FUNCTION_BLOCK FB_ConveyorPeerSequence IMPLEMENTS I_ConveyorSequence
VAR_INPUT

END_VAR
VAR_OUTPUT
END_VAR
VAR
	nStep : E_ConveyorPeerSequence;
END_VAR

METHOD M_ConveyorAction : BOOL
VAR_INPUT
	in_stFirstMessage : ST_Message;
	in_stMessageToCheckFor : ST_Message;
	in_stSecondMessage : ST_Message;
	in_rConveyor : REFERENCE TO FB_Conveyor;
END_VAR
VAR_INST
	nConveyorActionStep : UINT;
END_VAR
CASE nConveyorActionStep OF
	
	0:
		IF 	in_rConveyor.M_SendMessage
			(	
				in_stFirstMessage
			) 
			= E_PeerReturnCode.eMESSAGE_IN_OUTBOX 
			THEN
			
			nConveyorActionStep := 10;
			
		END_IF
		
	10:
		
	
		IF 	in_rConveyor.M_CompareMessageAndEmptyMailbox
			(	
				in_stMessageToCheckFor
			) 
			= E_PeerReturnCode.eMATCH_FOUND 
			THEN
			
			nConveyorActionStep := 20;
			
		END_IF

	20:
		
		IF 	in_rConveyor.M_SendMessage
			(	
				in_stSecondMessage
			) 
			= E_PeerReturnCode.eMESSAGE_IN_OUTBOX 
			THEN
			
			nConveyorActionStep := 0;
			M_ConveyorAction := TRUE;
			
		END_IF
		
END_CASE
END_METHOD


METHOD M_ConveyorSequence : BOOL
VAR_INPUT
	in_rConveyor : REFERENCE TO FB_Conveyor;
END_VAR
CASE nStep OF
	
	E_ConveyorPeerSequence.eSTOP:
	
		nStep := E_ConveyorPeerSequence.eSTART;
		
	E_ConveyorPeerSequence.eSTART:
		
		in_rConveyor.M_StartConveyor();
		nStep := E_ConveyorPeerSequence.eSTOP_AT_SIGNAL;

	E_ConveyorPeerSequence.eSTOP_AT_SIGNAL:
	
		IF in_rConveyor.out_fbSensorStop.GetSignal THEN
			in_rConveyor.M_StopConveyor();
			nStep := E_ConveyorPeerSequence.eWAIT_FOR_ACK;
		END_IF
	
	E_ConveyorPeerSequence.eWAIT_FOR_ACK:
		
		IF M_SubjectiveAction(in_rConveyor) THEN
			nStep := E_ConveyorPeerSequence.eRESUME_OPERATION;
		END_IF
	
	E_ConveyorPeerSequence.eRESUME_OPERATION:
		
		in_rConveyor.M_StartConveyor();
		IF in_rConveyor.out_fbSensorMaterialDispatch.GetSignal THEN
			in_rConveyor.M_StopConveyor();
			nStep := E_ConveyorPeerSequence.eEND_SEQUENCE;
		END_IF
	
	E_ConveyorPeerSequence.eEND_SEQUENCE:
		;
		
END_CASE
END_METHOD

METHOD M_Sequence : BOOL
VAR_INPUT
END_VAR
END_METHOD

METHOD M_SubjectiveAction : BOOL
VAR_INPUT
	in_rConveyor : REFERENCE TO FB_Conveyor;
END_VAR
CASE in_rConveyor.M_GetPeerId() OF

	E_PeersList.ePEER_CONVEYOR_1:
		
		IF 	M_ConveyorAction
			(
				Message(eCONVEYOR_1_AT_TRANSFER_POINT,ePEER_CONVEYOR_2),
				Message(eCONVEYOR_4_AT_TRANSFER_POINT,ePEER_CONVEYOR_4),
 				Message(eCONVEYOR_1_RESUMING_OPERATION,ePEER_CONVEYOR_2),
				in_rConveyor
			) 
			THEN
			
			M_SubjectiveAction := TRUE;
			
		END_IF
		
		
	E_PeersList.ePEER_CONVEYOR_2:

		IF 	M_ConveyorAction
			(
				Message(eCONVEYOR_2_AT_TRANSFER_POINT,ePEER_CONVEYOR_3),
				Message(eCONVEYOR_1_RESUMING_OPERATION,ePEER_CONVEYOR_1),
 				Message(eCONVEYOR_2_RESUMING_OPERATION,ePEER_CONVEYOR_3),
				in_rConveyor
			) 
			THEN
			
			M_SubjectiveAction := TRUE;
			
		END_IF	
	
	E_PeersList.ePEER_CONVEYOR_3:

		IF 	M_ConveyorAction
			(
				Message(eCONVEYOR_3_AT_TRANSFER_POINT,ePEER_CONVEYOR_4),
				Message(eCONVEYOR_2_RESUMING_OPERATION,ePEER_CONVEYOR_2),
 				Message(eCONVEYOR_3_RESUMING_OPERATION,ePEER_CONVEYOR_4),
				in_rConveyor
			) 
			THEN
			
			M_SubjectiveAction := TRUE;
			
		END_IF
	
	E_PeersList.ePEER_CONVEYOR_4:
	
		IF 	M_ConveyorAction
			(
				Message(eCONVEYOR_1_AT_TRANSFER_POINT,ePEER_CONVEYOR_2),
				Message(eCONVEYOR_3_RESUMING_OPERATION,ePEER_CONVEYOR_3),
 				Message(NULL,NULL),
				in_rConveyor
			) 
			THEN
			
			M_SubjectiveAction := TRUE;
			
		END_IF	

END_CASE
END_METHOD

END_FUNCTION_BLOCK

(* stored: Version 1.1.0.1, ProductVersion 3.1.4024.0
   POU FB_ConveyorPeerSequence: Id {9535a82b-99de-4536-9474-8a23e333c65a}, SpecialFunc None
   Method M_ConveyorAction: Id {9cd03c54-3668-4377-af34-5b4f618835e8}
   Method M_ConveyorSequence: Id {57fbfd93-eff7-400b-9875-503f49d69ce5}
   Method M_Sequence: Id {dab0eca6-3cd4-4ce7-9021-f50597f8cead}
   Method M_SubjectiveAction: Id {b3807608-e155-4afb-a89a-458a50a4675f} *)
